PROGRAM Axis02_Command
VAR
//System_Bit
	Always_ON	:	BOOL	:=TRUE	;//상시 ON 
	Always_OFF	:	BOOL	:=FALSE	;//상시 OFF

//Motor_Command
	Axis02: AXIS_REF;											//회전축
	Axis02_MC_Power: MC_Power;
	Axis02_MC_Home: FB_HomeBeforeMoveAX8000:=(channel:=2);
	Axis02_Jog: MC_Jog;
	Axis02_Home_Pos_Move: MC_MoveAbsolute;
	Axis02_Wait_Pos_Move: MC_MoveAbsolute;
	Axis02_Target_Pos_Move: MC_MoveAbsolute;
	Axi02_Work_End_Move: MC_GearInVelo;
	Work_Offset_Move: MC_MoveSuperImposed;
	Axis02_Work_End_Comp: MC_GearOut;
	Axis02_Maint_Move: MC_MoveAbsolute;
	Axis02_Tool_Change: MC_MoveAbsolute;
	Axis02_Calibration: MC_MoveAbsolute;	



	
	Test002: BOOL;
	Test001: BOOL;

	Axis02_Stop_02: MC_Stop;
	Work_Comp: BOOL;
	Work_Stop: BOOL;


	Timer01: TON;
	Axis02_Work_End_Move_Test: MC_MoveAbsolute;
	Encoder_Real_Velocity: LREAL;
	MC_GearInPos_0: MC_GearInPos;
END_VAR
VAR // added by the converter: edge detectors and wires of the graphical bodies
    _rt1, _rt2 : R_TRIG;
END_VAR

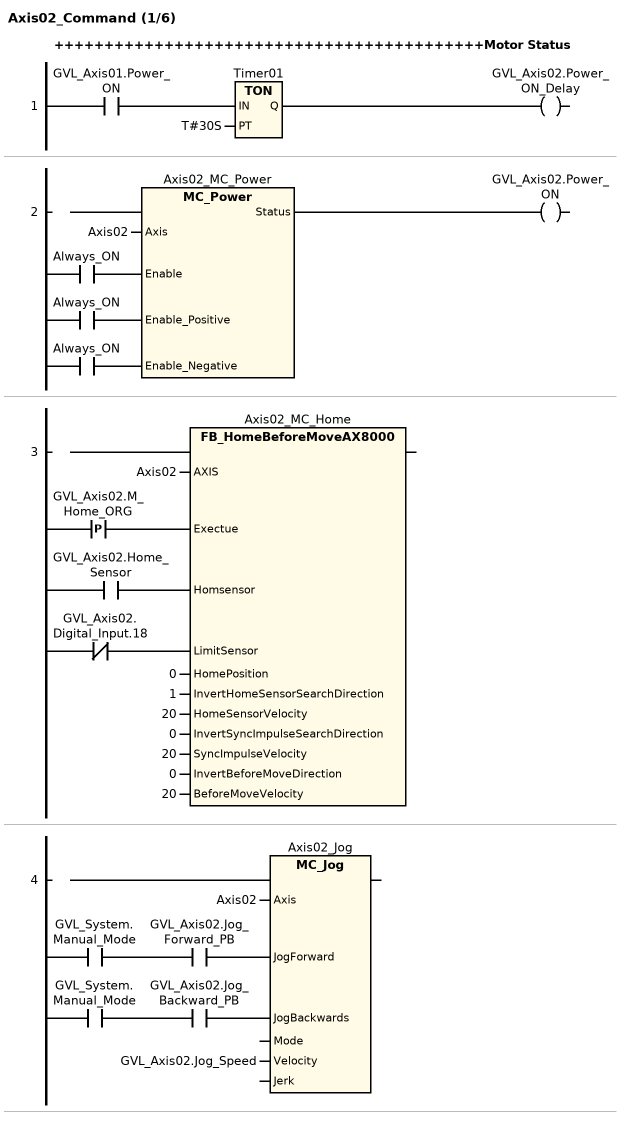
// NETWORK 1: +++++++++++++++++++++++++++++++++++++++++++Motor Status
Timer01(IN := GVL_Axis01.Power_ON, PT := T#30S); // TON
GVL_Axis02.Power_ON_Delay := Timer01.Q;

// NETWORK 2
Axis02_MC_Power(
    Axis := Axis02,
    Enable := Always_ON,
    Enable_Positive := Always_ON,
    Enable_Negative := Always_ON); // MC_Power
GVL_Axis02.Power_ON := Axis02_MC_Power.Status;

// NETWORK 3
_rt1(CLK := GVL_Axis02.M_Home_ORG);
Axis02_MC_Home(
    AXIS := Axis02,
    Exectue := _rt1.Q,
    Homsensor := GVL_Axis02.Home_Sensor,
    LimitSensor := NOT GVL_Axis02.Digital_Input.18,
    HomePosition := 0,
    InvertHomeSensorSearchDirection := 1,
    HomeSensorVelocity := 20,
    InvertSyncImpulseSearchDirection := 0,
    SyncImpulseVelocity := 20,
    InvertBeforeMoveDirection := 0,
    BeforeMoveVelocity := 20); // FB_HomeBeforeMoveAX8000

// NETWORK 4
Axis02_Jog(
    Axis := Axis02,
    JogForward := GVL_System.Manual_Mode AND GVL_Axis02.Jog_Forward_PB,
    JogBackwards := GVL_System.Manual_Mode AND GVL_Axis02.Jog_Backward_PB,
    Velocity := GVL_Axis02.Jog_Speed); // MC_Jog

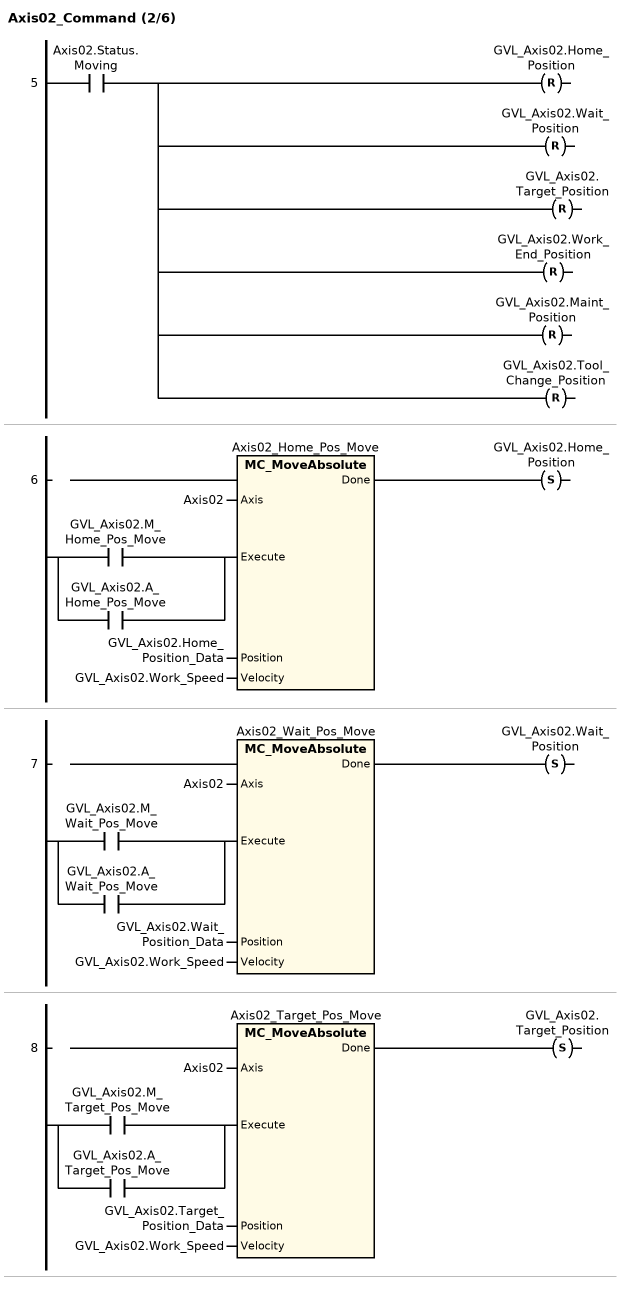
// NETWORK 5
GVL_Axis02.Home_Position R= Axis02.Status.Moving;
GVL_Axis02.Wait_Position R= Axis02.Status.Moving;
GVL_Axis02.Target_Position R= Axis02.Status.Moving;
GVL_Axis02.Work_End_Position R= Axis02.Status.Moving;
GVL_Axis02.Maint_Position R= Axis02.Status.Moving;
GVL_Axis02.Tool_Change_Position R= Axis02.Status.Moving;

// NETWORK 6
Axis02_Home_Pos_Move(
    Axis := Axis02,
    Execute := GVL_Axis02.M_Home_Pos_Move OR GVL_Axis02.A_Home_Pos_Move,
    Position := GVL_Axis02.Home_Position_Data,
    Velocity := GVL_Axis02.Work_Speed); // MC_MoveAbsolute
GVL_Axis02.Home_Position S= Axis02_Home_Pos_Move.Done;

// NETWORK 7
Axis02_Wait_Pos_Move(
    Axis := Axis02,
    Execute := GVL_Axis02.M_Wait_Pos_Move OR GVL_Axis02.A_Wait_Pos_Move,
    Position := GVL_Axis02.Wait_Position_Data,
    Velocity := GVL_Axis02.Work_Speed); // MC_MoveAbsolute
GVL_Axis02.Wait_Position S= Axis02_Wait_Pos_Move.Done;

// NETWORK 8
Axis02_Target_Pos_Move(
    Axis := Axis02,
    Execute := GVL_Axis02.M_Target_Pos_Move OR GVL_Axis02.A_Target_Pos_Move,
    Position := GVL_Axis02.Target_Position_Data,
    Velocity := GVL_Axis02.Work_Speed); // MC_MoveAbsolute
GVL_Axis02.Target_Position S= Axis02_Target_Pos_Move.Done;

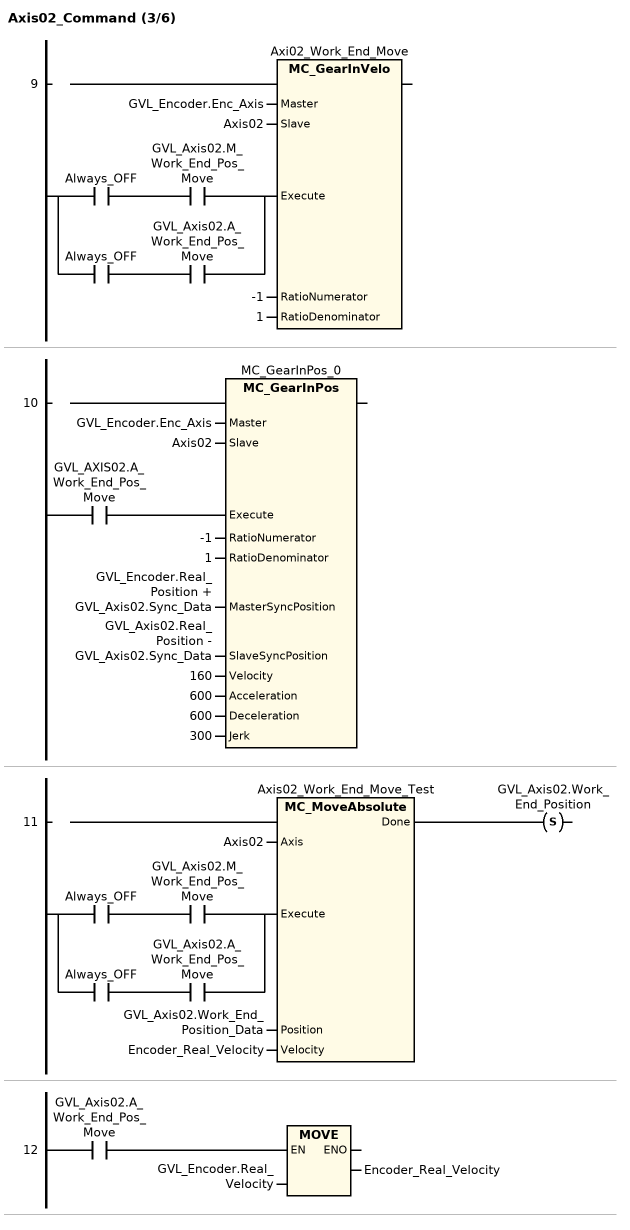
// NETWORK 9
Axi02_Work_End_Move(
    Master := GVL_Encoder.Enc_Axis,
    Slave := Axis02,
    Execute := Always_OFF AND GVL_Axis02.M_Work_End_Pos_Move OR Always_OFF AND GVL_Axis02.A_Work_End_Pos_Move,
    RatioNumerator := -1,
    RatioDenominator := 1); // MC_GearInVelo

// NETWORK 10
MC_GearInPos_0(
    Master := GVL_Encoder.Enc_Axis,
    Slave := Axis02,
    Execute := GVL_AXIS02.A_Work_End_Pos_Move,
    RatioNumerator := -1,
    RatioDenominator := 1,
    MasterSyncPosition := GVL_Encoder.Real_Position + GVL_Axis02.Sync_Data,
    SlaveSyncPosition := GVL_Axis02.Real_Position - GVL_Axis02.Sync_Data,
    Velocity := 160,
    Acceleration := 600,
    Deceleration := 600,
    Jerk := 300); // MC_GearInPos

// NETWORK 11
Axis02_Work_End_Move_Test(
    Axis := Axis02,
    Execute := Always_OFF AND GVL_Axis02.M_Work_End_Pos_Move OR Always_OFF AND GVL_Axis02.A_Work_End_Pos_Move,
    Position := GVL_Axis02.Work_End_Position_Data,
    Velocity := Encoder_Real_Velocity); // MC_MoveAbsolute
GVL_Axis02.Work_End_Position S= Axis02_Work_End_Move_Test.Done;

// NETWORK 12
IF GVL_Axis02.A_Work_End_Pos_Move THEN Encoder_Real_Velocity := GVL_Encoder.Real_Velocity; END_IF

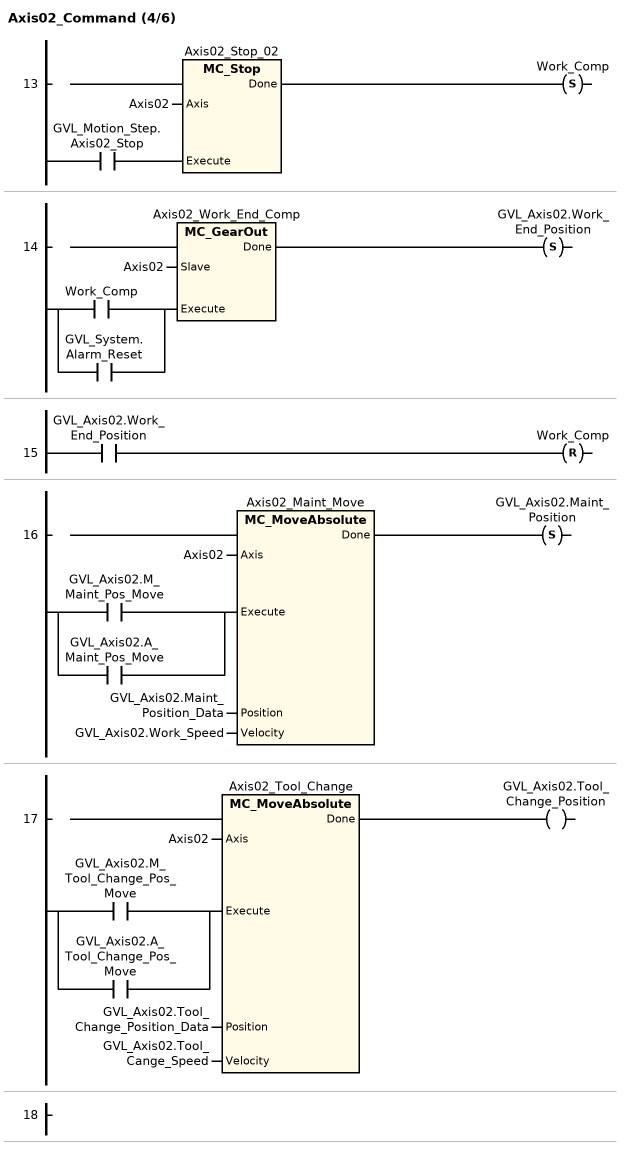
// NETWORK 13
Axis02_Stop_02(Axis := Axis02, Execute := GVL_Motion_Step.Axis02_Stop); // MC_Stop
Work_Comp S= Axis02_Stop_02.Done;

// NETWORK 14
Axis02_Work_End_Comp(Slave := Axis02, Execute := Work_Comp OR GVL_System.Alarm_Reset); // MC_GearOut
GVL_Axis02.Work_End_Position S= Axis02_Work_End_Comp.Done;

// NETWORK 15
Work_Comp R= GVL_Axis02.Work_End_Position;

// NETWORK 16
Axis02_Maint_Move(
    Axis := Axis02,
    Execute := GVL_Axis02.M_Maint_Pos_Move OR GVL_Axis02.A_Maint_Pos_Move,
    Position := GVL_Axis02.Maint_Position_Data,
    Velocity := GVL_Axis02.Work_Speed); // MC_MoveAbsolute
GVL_Axis02.Maint_Position S= Axis02_Maint_Move.Done;

// NETWORK 17
Axis02_Tool_Change(
    Axis := Axis02,
    Execute := GVL_Axis02.M_Tool_Change_Pos_Move OR GVL_Axis02.A_Tool_Change_Pos_Move,
    Position := GVL_Axis02.Tool_Change_Position_Data,
    Velocity := GVL_Axis02.Tool_Cange_Speed); // MC_MoveAbsolute
GVL_Axis02.Tool_Change_Position := Axis02_Tool_Change.Done;

// NETWORK 18

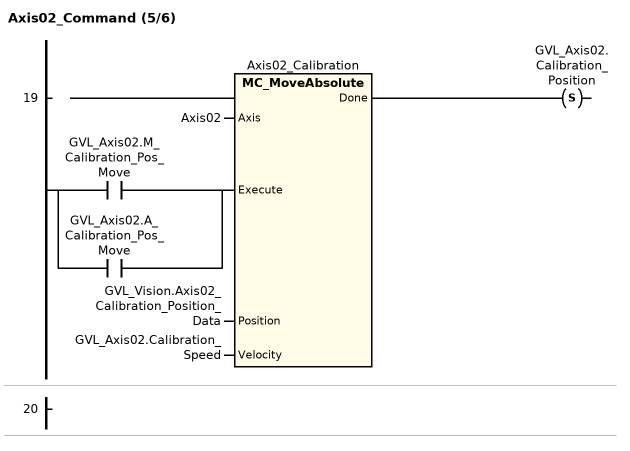
// NETWORK 19
Axis02_Calibration(
    Axis := Axis02,
    Execute := GVL_Axis02.M_Calibration_Pos_Move OR GVL_Axis02.A_Calibration_Pos_Move,
    Position := GVL_Vision.Axis02_Calibration_Position_Data,
    Velocity := GVL_Axis02.Calibration_Speed); // MC_MoveAbsolute
GVL_Axis02.Calibration_Position S= Axis02_Calibration.Done;

// NETWORK 20

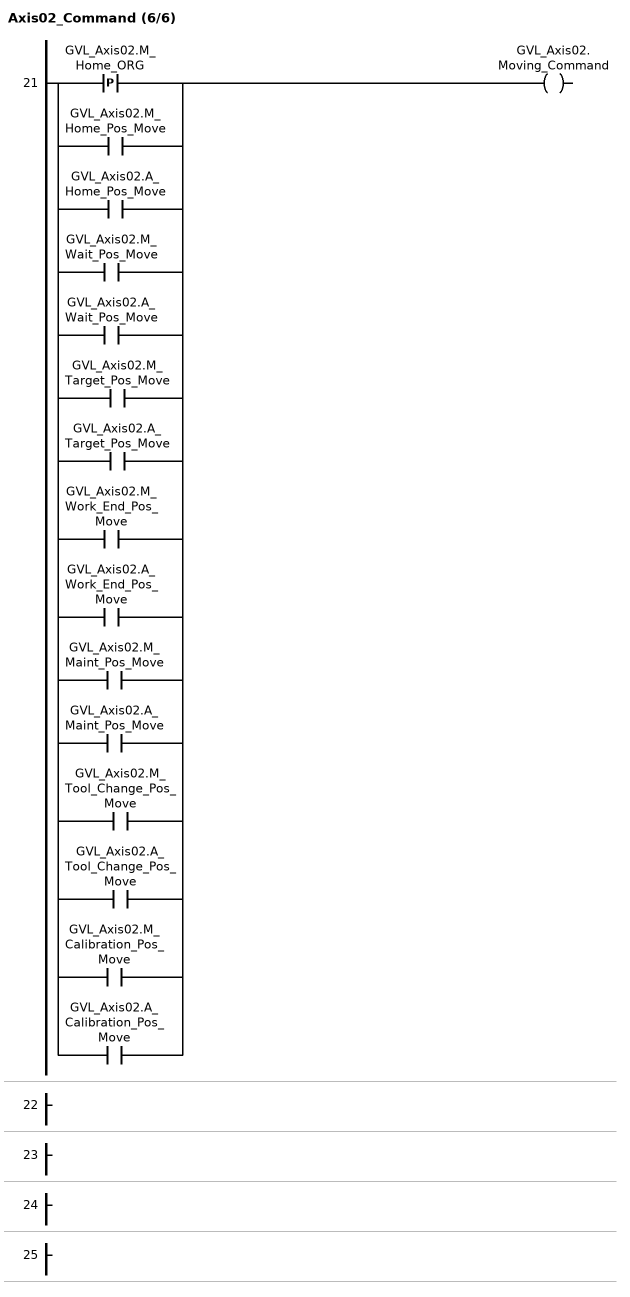
// NETWORK 21
_rt2(CLK := GVL_Axis02.M_Home_ORG);
GVL_Axis02.Moving_Command := _rt2.Q OR GVL_Axis02.M_Home_Pos_Move OR GVL_Axis02.A_Home_Pos_Move OR GVL_Axis02.M_Wait_Pos_Move OR GVL_Axis02.A_Wait_Pos_Move OR GVL_Axis02.M_Target_Pos_Move OR GVL_Axis02.A_Target_Pos_Move OR GVL_Axis02.M_Work_End_Pos_Move OR GVL_Axis02.A_Work_End_Pos_Move OR GVL_Axis02.M_Maint_Pos_Move OR GVL_Axis02.A_Maint_Pos_Move OR GVL_Axis02.M_Tool_Change_Pos_Move OR GVL_Axis02.A_Tool_Change_Pos_Move OR GVL_Axis02.M_Calibration_Pos_Move OR GVL_Axis02.A_Calibration_Pos_Move;

// NETWORK 22

// NETWORK 23

// NETWORK 24

// NETWORK 25

END_PROGRAM

(* stored: Version 1.1.0.1, ProductVersion 3.1.4024.15
   POU Axis02_Command: Id {abb82378-bf1f-48b6-8374-4c4feca42d94}, SpecialFunc None *)
